TYPE ST_TimeManagement_SP :
STRUCT
	TotalUpTime				: ST_ElapsedTime;	//Total up time of System
	PreviousDay				: INT;				//Previous day, used for midnight pulse
END_STRUCT
END_TYPE

(* stored: Version 1.1.0.1, ProductVersion 3.1.4024.2
   DUT ST_TimeManagement_SP: Id {e8f31541-6351-4ef2-af5d-64a3c1f7f964} *)
